FUNCTION BYTE_TO_ARR08X (* this Function extracts the 8 BOOLS from a byte and make a 8-BOOL Array *)
  (* Standard: 61499-1; Description: Copyright (c) 2024 HR Agrartechnik GmbH This program and the accompanying materials are made available under the terms of the Eclipse Public License 2.0 which is available at https://www.eclipse.org/legal/epl-2.0/ SPDX-License-Identifier: EPL-2.0 *)
  (* Version 1.0, 2024-02-22, Franz Höpfinger, HR Agrartechnik GmbH *)
  PACKAGE logiBUS::utils::conversion::arr::splitting;
  IMPORT eclipse4diac::core::TypeHash;
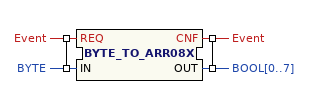
  EVENT_INPUT
    REQ WITH IN;
  END_EVENT
  EVENT_OUTPUT
    CNF WITH OUT;
  END_EVENT
  VAR_INPUT
    IN : BYTE; (* BYTE Input *)
  END_VAR
  VAR_OUTPUT
    OUT : ARRAY [0..7] OF BOOL; (* ARR08B Output *)
  END_VAR
  BODY IN ST:
PACKAGE logiBUS::utils::conversion::arr::splitting;

(* this Function extracts the 8 BOOLS from a byte and make a 8-BOOL Array *)
FUNCTION BYTE_TO_ARR08X

VAR_INPUT
	IN : BYTE; // BYTE Input
END_VAR

VAR_OUTPUT
	OUT : ARRAY[0..7] OF BOOL; // ARR08B Output
END_VAR

OUT[0] := IN.0;
OUT[1] := IN.1;
OUT[2] := IN.2;
OUT[3] := IN.3;
OUT[4] := IN.4;
OUT[5] := IN.5;
OUT[6] := IN.6;
OUT[7] := IN.7;

END_FUNCTION
  END_BODY
END_FUNCTION
